# B&R Automation Studio project CombinedLinenSoiledA9KAN (part 8)

#### mnEthInit.st - Initialization code
```iecst
(********************************************************************
 * COPYRIGHT --
 ********************************************************************
 * Program: mnEth
 * File: mnEthInit.st
 * Author: hunholz
 * Created: August 9, 2011
 * Changed: February 3, 2012 2.07.0
 ********************************************************************
 * Implementation of program mnEth
 ********************************************************************)

PROGRAM _INIT

	_xmnEthOk := TRUE;

	_xDHCPstarted := FALSE;
	_xSNTPSrvStarted := FALSE;
	_xSNTPCltStarted := FALSE;

	brsmemset(ADR(kgMsgStatus[MNETH_IDX_KGMSGSTAT]),0,SIZEOF(kgMsgStatus[0]));

	kgMsgStatus[MNETH_IDX_KGMSGSTAT].wFunction_ID := 4;

	// Packet-Version auslesen mit MO_ver aus SYS_lib und für den Additional Status zur Verfügung stellen

	_sPkgName := 'mnEth';

	IF ( MO_ver(ADR(_sPkgName), 0, ADR(_VerStruc)) = 0 ) THEN

		brsmemcpy(ADR(mnEthStatAd.sPkgVersion), ADR(_VerStruc.version), SIZEOF(_VerStruc.version));

	ELSE

		mnEthStatAd.sPkgVersion := '---';

	END_IF

	//***********************************************
	//Lese das Ethernet-Device der CPU aus
	//***********************************************
	REPEAT

		_GetEthPort(enable := TRUE, adrIF := ADR(_sEthDevice));

	UNTIL

		_GetEthPort.status <> ERR_FUB_BUSY

	END_REPEAT

//	brsstrcpy(ADR(_sEthDevice),ADR('IF2'));

		IF brsstrcmp(ADR(_sEthDevice), ADR('ERR')) = 0 THEN

		kgMsgStatus[MNETH_IDX_KGMSGSTAT].wMsgAckLevel := 0;
		kgMsgStatus[MNETH_IDX_KGMSGSTAT].wMsgClass := 10;
		kgMsgStatus[MNETH_IDX_KGMSGSTAT].wMsgNumber := _MENETH_MSG_IFDEVICE;

		_xmnEthOk := FALSE;
		ZANE[1]:= 1;
	END_IF

	//**********************************************************
	//Bestimme den Hostnamen der SPS und setze ihn
	//**********************************************************

	// Adresse von _Info_.InfoGeneral.utfMaschinennummer suchen

//	_xInfoExist := PV_xgetadr(ADR('_Info_.InfoGeneral.utfMaschinennummer'), ADR(_pInfoMaschinennummer), ADR(_lLenInfoMaschinennummer)) = ERR_OK;
//	_xInfoExist := _xInfoExist AND (_lLenInfoMaschinennummer >= 32);

	_xSetDefault := FALSE;

	_CfgGetInaNode(enable := TRUE, pDevice := ADR(_sEthDevice));

	IF _CfgGetInaNode.status = ERR_OK THEN

		IF _CfgGetInaNode.InaNode = 16#FE THEN

			// Setze auf jeden Fall die Default Adresse
			_xSetDefault := TRUE;

		END_IF

	END_IF

	//********************************************************************************************
	//Erzeuge einen Speicherbereich zum parsen oder schreiben von CSV-Dateien
	//********************************************************************************************

	_pParseMem := 0;

	_MemPartCreate(enable := TRUE, len := 512);

	IF _MemPartCreate.status = ERR_OK THEN

		_MemPartAlloc(enable := TRUE, ident := _MemPartCreate.ident, len := 256);

		IF _MemPartAlloc.status = ERR_OK THEN

			_pParseMem := _MemPartAlloc.mem;

		ELSE

			kgMsgStatus[MNETH_IDX_KGMSGSTAT].wMsgAckLevel := 0;
			kgMsgStatus[MNETH_IDX_KGMSGSTAT].wMsgClass := 10;
			kgMsgStatus[MNETH_IDX_KGMSGSTAT].wMsgNumber := _MENETH_MSG_MEM;

			_xmnEthOk := FALSE;
			ZANE[3] := 1;
		END_IF

	ELSE

		kgMsgStatus[MNETH_IDX_KGMSGSTAT].wMsgAckLevel := 0;
		kgMsgStatus[MNETH_IDX_KGMSGSTAT].wMsgClass := 10;
		kgMsgStatus[MNETH_IDX_KGMSGSTAT].wMsgNumber := _MENETH_MSG_MEM;

		_xmnEthOk := FALSE;
	ZANE[2] := 1;

	END_IF

	//**********************************************************
	// Prüfe, ob ein USB-Speicher gesteckt ist
	//**********************************************************

//	_xUSBexist := FALSE;
//
//	IF _xmnEthOk THEN
//
//		_UsbNodeListGet(enable := TRUE, pBuffer := ADR(_NodeIdBuffer), bufferSize := SIZEOF(_NodeIdBuffer), filterInterfaceClass := asusb_CLASS_MASS_STORAGE, filterInterfaceSubClass := 0);
//
//		IF _UsbNodeListGet.status = ERR_OK THEN
//
//			IF _UsbNodeListGet.listNodes > 0 THEN
//
//				_UsbNodeGet(enable := TRUE, nodeId := _NodeIdBuffer[0], pBuffer := ADR(_UsbBufferData), bufferSize := SIZEOF(_UsbBufferData));
//
//				IF _UsbNodeGet.status = ERR_OK THEN
//
//					_sUSBDeviceString := '/DEVICE=';
//					brsstrcpy(ADR(_sUSBDeviceString), ADR(_UsbBufferData.ifName));
//					_xUSBexist := TRUE;
//
//				END_IF
//
//			END_IF
//
//		END_IF
//
//	END_IF

	//******************************************************************************
	// Wenn nicht default gesetzt werden soll, csv-Datei auf USB suchen
	//******************************************************************************

	_xSetIPFromUsb := FALSE;

	IF _xmnEthOk THEN

		IF NOT _xSetDefault THEN

			brsstrcpy(ADR(_sPathCsv), ADR(_sHostname));
			brsstrcat(ADR(_sPathCsv), ADR('\mnEth\mnEth.csv'));

			_FileOpenCsv(enable := TRUE, pDevice := ADR(KG_DEVICE_USBSTICK1), pFile := ADR(_sPathCsv), mode := fiREAD_ONLY);

			IF _FileOpenCsv.status <> ERR_OK THEN

				_FileOpenCsv(enable := TRUE, pDevice := ADR(KG_DEVICE_USBSTICK2), pFile := ADR(_sPathCsv), mode := fiREAD_ONLY);

			END_IF

			IF _FileOpenCsv.status = ERR_OK THEN

				_FileReadCsv(enable := TRUE, ident := _FileOpenCsv.ident, pDest := _pParseMem, len := 256);

				IF _FileReadCsv.status = ERR_OK THEN

					_GetCsvDat.enable := TRUE;
					brwcsncpy( ADR(_GetCsvDat.utfCsvString), _pParseMem+2, 126);
					_GetCsvDat();

					IF _GetCsvDat.RowType = 90 THEN

						brwcsconv(ADR(_ParSetUsb.IP_Adr), ADR(_GetCsvDat.CsvIPRow.utfIP_Adress), 1);
						brwcsconv(ADR(_ParSetUsb.Gateway_Adr), ADR(_GetCsvDat.CsvIPRow.utfGateway), 1);

						IF ethInetAton(pIpStr := ADR(_ParSetUsb.IP_Adr), ADR(_lIPAdr)) = ERR_OK THEN

							IF ethInetAton(pIpStr := ADR(_ParSetUsb.Gateway_Adr), ADR(_lGatewayAdr)) = ERR_OK THEN

								_pOctet ACCESS ADR(_lIPAdr);

								_ParSetUsb.IP_ID1 := _pOctet[0];
								_ParSetUsb.IP_ID2 := _pOctet[1];
								_ParSetUsb.IP_ID3 := (_pOctet[2] / 16) * 16;
								_ParSetUsb.Region := _pOctet[2] MOD 16;
								_ParSetUsb.Station := _pOctet[3];

								IF _ParSetUsb.Region = 3 THEN
									_ParSetUsb.Number := kgGetLineNumberW3(Station := _ParSetUsb.Station, pMachineType := ADR(_kgMachineTypeW3));
								ELSE
									_ParSetUsb.Number := 0;
								END_IF

								// NET-Id bestimmen
								_lNetId := _lIPAdr;
								_pOctet ACCESS ADR(_lNetId);

								_pOctet[2] := _ParSetUsb.IP_ID3;
								_pOctet[3] := 0;

								ethInetNtoa(ipAdr := _lNetId, pIpStr := ADR(_ParSetUsb.NetId_Adr));

								_pOctet ACCESS ADR(_lGatewayAdr);

								_ParSetUsb.GW_ID1 := _pOctet[0];
								_ParSetUsb.GW_ID2 := _pOctet[1];
								_ParSetUsb.GW_ID3 := _pOctet[2];
								_ParSetUsb.GW_ID4 := _pOctet[3];

								_xSetIPFromUsb := TRUE;

							END_IF

						END_IF

					END_IF

				END_IF

				_FileCloseCsv(enable := TRUE, ident := _FileOpenCsv.ident);

			END_IF

//			_sParam := '/DEVICE=';
//			brsstrcat(ADR(_sParam), ADR(_sUSBDeviceString));
//
//			_sUSBDeviceName := 'STICK';
//
//			_DeviceLink(enable := TRUE, pDevice := ADR(_sUSBDeviceName), pParam := ADR(_sParam));
//
//			IF _DeviceLink.status = ERR_OK  AND _pParseMem <> 0 THEN
//
//				_FileOpenCsv(enable := TRUE, pDevice := ADR(_sUSBDeviceName), pFile := ADR(_sPathCsv), mode := fiREAD_ONLY);
//
//				IF _FileOpenCsv.status = ERR_OK THEN
//
//					_FileReadCsv(enable := TRUE, ident := _FileOpenCsv.ident, pDest := _pParseMem, len := 256);
//
//					IF _FileReadCsv.status = ERR_OK THEN
//
//						_GetCsvDat.enable := TRUE;
//						brwcsncpy( ADR(_GetCsvDat.utfCsvString), _pParseMem+2, 126);
//						_GetCsvDat();
//
//						IF _GetCsvDat.RowType = 90 THEN
//
//							brwcsconv(ADR(_ParSetUsb.IP_Adr), ADR(_GetCsvDat.CsvIPRow.utfIP_Adress), 1);
//							brwcsconv(ADR(_ParSetUsb.Gateway_Adr), ADR(_GetCsvDat.CsvIPRow.utfGateway), 1);
//
//							IF ethInetAton(pIpStr := ADR(_ParSetUsb.IP_Adr), ADR(_lIPAdr)) = ERR_OK THEN
//
//								IF ethInetAton(pIpStr := ADR(_ParSetUsb.Gateway_Adr), ADR(_lGatewayAdr)) = ERR_OK THEN
//
//									_pOctet ACCESS ADR(_lIPAdr);
//
//									_ParSetUsb.IP_ID1 := _pOctet[0];
//									_ParSetUsb.IP_ID2 := _pOctet[1];
//									_ParSetUsb.IP_ID3 := (_pOctet[2] / 16) * 16;
//									_ParSetUsb.Region := _pOctet[2] MOD 16;
//									_ParSetUsb.Station := _pOctet[3];
//
//									IF _ParSetUsb.Region = 3 THEN
//										_ParSetUsb.Number := kgGetMachinenumberW3(Station := _ParSetUsb.Station, pMachineType := ADR(_kgMachineTypeW3));
//									ELSE
//										_ParSetUsb.Number := 0;
//									END_IF
//
//									// NET-Id bestimmen
//									_lNetId := _lIPAdr;
//									_pOctet ACCESS ADR(_lNetId);
//
//									_pOctet[2] := _ParSetUsb.IP_ID3;
//									_pOctet[3] := 0;
//
//									ethInetNtoa(ipAdr := _lNetId, pIpStr := ADR(_ParSetUsb.NetId_Adr));
//
//									_pOctet ACCESS ADR(_lGatewayAdr);
//
//									_ParSetUsb.GW_ID1 := _pOctet[0];
//									_ParSetUsb.GW_ID2 := _pOctet[1];
//									_ParSetUsb.GW_ID3 := _pOctet[2];
//									_ParSetUsb.GW_ID4 := _pOctet[3];
//
//									_xSetIPFromUsb := TRUE;
//
//								END_IF
//
//							END_IF
//
//						END_IF
//
//					END_IF
//
//					_FileCloseCsv(enable := TRUE, ident := _FileOpenCsv.ident);
//
//				END_IF
//
//				_DeviceUnlink(enable := TRUE, handle := _DeviceLink.handle);
//
//			END_IF

		END_IF

	END_IF

	//********************************************************************************
	// Sicherstellen, dass das Verzeichnis mnEth auf der CF-Card existiert
	//********************************************************************************

	_DirInfo(enable := TRUE, pDevice := ADR(KG_DEVICE_COMPACTFLASH), pPath := ADR('mnEth'));

	IF _DirInfo.status <> ERR_OK THEN

		_DirCreate(enable := TRUE, pDevice := ADR(KG_DEVICE_COMPACTFLASH), pName := ADR('mnEth'));

	END_IF

	//*****************************************************************************************************
	// Wenn nicht default und nicht von USB gesetzt werden soll, csv-Datei auf CF suchen
	//*****************************************************************************************************

	_xSetIPFromCF := FALSE;

	_sPathCsv := 'mnEth\mnEth.csv';

	IF _xmnEthOk THEN

		IF NOT _xSetDefault  AND NOT _xSetIPFromUsb THEN

			_sPathCsv := 'mnEth\mnEth.csv';

			_FileOpenCsv(enable := TRUE, pDevice := ADR(KG_DEVICE_COMPACTFLASH), pFile := ADR(_sPathCsv), mode := fiREAD_ONLY);

			IF _FileOpenCsv.status = ERR_OK THEN

				_FileReadCsv(enable := TRUE, ident := _FileOpenCsv.ident, pDest := _pParseMem, len := 256);

				IF _FileReadCsv.status = ERR_OK THEN

					_GetCsvDat.enable := TRUE;
					brwcsncpy( ADR(_GetCsvDat.utfCsvString), _pParseMem+2, 126);
					// Nur erste Zeile
					_lPosLF := brwcschr(ADR(_GetCsvDat.utfCsvString),16#0A);
					_lPosCR := brwcschr(ADR(_GetCsvDat.utfCsvString),16#0D);
					IF (_lPosCR <> 0) THEN
						brsmemset(_lPosCR , 0, 2);
					END_IF
					IF (_lPosLF <> 0) THEN
						brsmemset(_lPosLF , 0, 2);
					END_IF

					_GetCsvDat();

					IF _GetCsvDat.RowType = 90 THEN

						brwcsconv(ADR(_ParSetCF.IP_Adr), ADR(_GetCsvDat.CsvIPRow.utfIP_Adress), 1);
						brwcsconv(ADR(_ParSetCF.Gateway_Adr), ADR( _GetCsvDat.CsvIPRow.utfGateway), 1);

						IF ethInetAton(pIpStr := ADR(_ParSetCF.IP_Adr), ADR(_lIPAdr)) = ERR_OK THEN

							IF ethInetAton(pIpStr := ADR(_ParSetCF.Gateway_Adr), ADR(_lGatewayAdr)) = ERR_OK THEN

								_pOctet ACCESS ADR(_lIPAdr);

								_ParSetCF.IP_ID1 := _pOctet[0];
								_ParSetCF.IP_ID2 := _pOctet[1];
								_ParSetCF.IP_ID3 := (_pOctet[2] / 16) * 16;
								_ParSetCF.Region := _pOctet[2] MOD 16;
								_ParSetCF.Station := _pOctet[3];

								IF _ParSetCF.Region = 3 THEN
									_ParSetCF.Number := kgGetLineNumberW3(Station := _ParSetCF.Station, pMachineType := ADR(_kgMachineTypeW3));
								ELSE
									_ParSetCF.Number := 0;
								END_IF

								// NET-Id bestimmen
								_lNetId := _lIPAdr;
								_pOctet ACCESS ADR(_lNetId);

								_pOctet[2] := _ParSetCF.IP_ID3;
								_pOctet[3] := 0;

								ethInetNtoa(ipAdr := _lNetId, pIpStr := ADR(_ParSetCF.NetId_Adr));

								_pOctet ACCESS ADR(_lGatewayAdr);

								_ParSetCF.GW_ID1 := _pOctet[0];
								_ParSetCF.GW_ID2 := _pOctet[1];
								_ParSetCF.GW_ID3 := _pOctet[2];
								_ParSetCF.GW_ID4 := _pOctet[3];

								_xSetIPFromCF := TRUE;

							END_IF

						END_IF

					END_IF

				END_IF

				_FileCloseCsv(enable := TRUE, ident := _FileOpenCsv.ident);

			END_IF

		END_IF

	END_IF

	//*****************************************************************************************************
	// Adressen von CF oder USB setzen
	//*****************************************************************************************************

	IF _xmnEthOk THEN

		IF _xSetIPFromCF OR _xSetIPFromUsb THEN

			IF _xSetIPFromCF THEN
				_ParSet := _ParSetCF;
			ELSE
				_ParSet := _ParSetUsb;
			END_IF

// Für Testzwecke in Hausnetzen mit anderer Netzwerkmaske

#ifndef NoSubnetMask

			_CfgGetSubnetMask(enable := TRUE, pDevice := ADR(_sEthDevice), pSubnetMask := ADR(_sActSubnetMask), Len := SIZEOF(_sActSubnetMask));

			IF (brsstrcmp(ADR(_sActSubnetMask), ADR(_sSubnetMask)) <> 0) THEN

				_CfgSetSubnetMask(enable := TRUE, pDevice := ADR(_sEthDevice), pSubnetMask := ADR(_sSubnetMask), Option := cfgOPTION_NON_VOLATILE);

			END_IF
#endif
			_pOctet ACCESS ADR(_lBroadcastAdr);

			_pOctet[0] := _ParSet.IP_ID1;
			_pOctet[1] := _ParSet.IP_ID2;
			_pOctet[2] := _ParSet.IP_ID3 + 15;
			_pOctet[3] := 255;

			ethInetNtoa(ADR(_lBroadcastAdr), ADR(_sBroadcastAdr));

			_CfgGetBroadcastAdr(enable := TRUE, pDevice := ADR(_sEthDevice), pBroadcastAddr := ADR(_sActBroadcastAdr), Len := SIZEOF(_sActBroadcastAdr));

			IF (brsstrcmp(ADR(_sActBroadcastAdr), ADR(_sBroadcastAdr)) <> 0) THEN

				_CfgSetBroadcastAdr(enable := TRUE, pDevice := ADR(_sEthDevice), pBroadcastAddr := ADR(_sBroadcastAdr), Option := cfgOPTION_NON_VOLATILE);

			END_IF

			_CfgGetIPAddress(enable := TRUE, pDevice := ADR(_sEthDevice), pIPAddr := ADR(_sActIPAdr), Len := SIZEOF(_sActIPAdr));

			IF (brsstrcmp(ADR(_sActIPAdr), ADR(_ParSet.IP_Adr)) <> 0) THEN

				_CfgSetIPAddr(enable := TRUE, pDevice := ADR(_sEthDevice), pIPAddr := ADR(_ParSet.IP_Adr), Option := cfgOPTION_NON_VOLATILE);

			END_IF

			_CfgGetGateway(enable := TRUE, pDevice := ADR(_sEthDevice), pGateway := ADR(_sActGateway), Len := SIZEOF(_sActGateway));

			IF (brsstrcmp(ADR(_sActGateway), ADR(_ParSet.Gateway_Adr)) <> 0) THEN

				_CfgSetDefaultGateway(enable := TRUE, pDevice := ADR(_sEthDevice), pGateway := ADR(_ParSet.Gateway_Adr), Option := cfgOPTION_NON_VOLATILE);

			END_IF

			_ParAktuell := _ParSet;

		ELSE

			_CfgGetGateway(enable := TRUE, pDevice := ADR(_sEthDevice), pGateway := ADR(_ParAktuell.Gateway_Adr), Len := SIZEOF(_ParAktuell.Gateway_Adr));

			_CfgGetIPAddress(enable := TRUE, pDevice := ADR(_sEthDevice), pIPAddr := ADR(_ParAktuell.IP_Adr), Len := SIZEOF(_ParAktuell.IP_Adr));

			IF ethInetAton(pIpStr := ADR(_ParAktuell.IP_Adr), ADR(_lIPAdr)) = ERR_OK THEN

				IF ethInetAton(pIpStr := ADR(_ParAktuell.Gateway_Adr), ADR(_lGatewayAdr)) = ERR_OK THEN

					_pOctet ACCESS ADR(_lIPAdr);

					_ParAktuell.IP_ID1 := _pOctet[0];
					_ParAktuell.IP_ID2 := _pOctet[1];
					_ParAktuell.IP_ID3 := (_pOctet[2] / 16) * 16;
					_ParAktuell.Region := _pOctet[2] MOD 16;
					_ParAktuell.Station := _pOctet[3];

					IF _ParAktuell.Region = 3 THEN
						_ParAktuell.Number := kgGetLineNumberW3(Station := _ParAktuell.Station, pMachineType := ADR(_kgMachineTypeW3));
					ELSE
						_ParAktuell.Number := 0;
					END_IF

					// NET-Id bestimmen
					_lNetId := _lIPAdr;
					_pOctet ACCESS ADR(_lNetId);

					_pOctet[2] := _ParAktuell.IP_ID3;
					_pOctet[3] := 0;

					ethInetNtoa(ipAdr := _lNetId, pIpStr := ADR(_ParAktuell.NetId_Adr));

					_pOctet ACCESS ADR(_lGatewayAdr);

					_ParAktuell.GW_ID1 := _pOctet[0];
					_ParAktuell.GW_ID2 := _pOctet[1];
					_ParAktuell.GW_ID3 := _pOctet[2];
					_ParAktuell.GW_ID4 := _pOctet[3];

				END_IF

			END_IF

		END_IF

		IF NOT _xSetIPFromCF AND NOT _xSetIPFromUsb THEN

			_xSetDefault := TRUE;

		END_IF

		_xChanged := FALSE;

	END_IF

	//*****************************************************************************************************
	// CSV-Datei schreiben, wenn Daten vom USB gekommen sind
	//*****************************************************************************************************

	IF _xmnEthOk THEN

		IF _xSetIPFromUsb OR NOT _xSetIPFromCF THEN

			brsmemset(_pParseMem, 0, 256);

			_lFileSize := 0;

			brwcsconv(ADR( _IPRow.utfIP_Adress), ADR(_ParAktuell.IP_Adr), 0);
			brwcsconv(ADR(_IPRow.utfGateway), ADR(_ParAktuell.Gateway_Adr), 0);

			_WriteBOM(enable := TRUE, pMem := _pParseMem, lMaxSize := 256, lSize := _lFileSize);
			_WriteCsv90(enable := TRUE, pMem := _pParseMem, lMaxSize := 256, IPRow := _IPRow, lSize := _lFileSize);

			_FileDeleteCsv(enable := TRUE, pDevice := ADR(KG_DEVICE_COMPACTFLASH), pName := ADR(_sPathCsv));

			_FileCreateCsv(enable := TRUE, pDevice := ADR(KG_DEVICE_COMPACTFLASH), pFile := ADR(_sPathCsv));

			_FileOpenCsv(enable := TRUE, pDevice := ADR(KG_DEVICE_COMPACTFLASH), pFile := ADR(_sPathCsv), mode := fiWRITE_ONLY);

			IF _FileOpenCsv.status = ERR_OK THEN

				_FileWriteCsv(enable := TRUE, ident := _FileOpenCsv.ident, offset := 0, pSrc := _pParseMem, len := _lFileSize);

				_FileCloseCsv(enable := TRUE, ident := _FileOpenCsv.ident);

			END_IF

		END_IF

	END_IF

END_PROGRAM
```

#### mnEth.typ - Local data types
```iecst
(********************************************************************
 * COPYRIGHT --
 ********************************************************************
 * Program: mnEth
 * File: mnEth.typ
 * Author: tamme
 * Created: March 17, 2011
 ********************************************************************
 * Local data types of program mnEth
 ********************************************************************)

TYPE
	enumEthernetState :
		(
		es_idle := 0,
		es_SetDef1 := 100,
		es_SetDef2,
		es_SetDef3,
		es_SetDef4,
		es_SetDef5,
		es_WriteCSV1 := 200,
		es_WriteCSV2,
		es_WriteCSV3,
		es_WriteCSV4,
		es_WriteCSV5,
		es_WriteCSV6,
		es_Change1 := 300,
		es_Change2,
		es_Change3,
		es_Change4,
		es_Change5,
		es_Change6,
		es_Change7,
		es_DHCP1 := 400,
		es_DHCP2,
		es_DHCP3,
		es_SNTPcltStart1 := 500,
		es_SNTPcltStop1 := 510,
		es_SNTPsrvStart1 := 520,
		es_SNTPsrvStop1 := 530,
		es_SetHostname1 := 600,
		es_SetHostname2,
		es_SetHostname3,
		es_Warning := 900
		);
	_EthPar_typ : 	STRUCT
		IP_ID1 : USINT;
		IP_ID2 : USINT;
		IP_ID3 : USINT;
		Region : USINT;
		Station : USINT;
		Number : USINT;
		GW_ID1 : USINT;
		GW_ID2 : USINT;
		GW_ID3 : USINT;
		GW_ID4 : USINT;
		IP_Adr : STRING[15];
		Gateway_Adr : STRING[15];
		NetId_Adr : STRING[15];
	END_STRUCT;
END_TYPE
```

#### mnEth.var - Local variables
```iecst
(********************************************************************
 * COPYRIGHT --
 ********************************************************************
 * Program: mnEth
 * File: mnEth.var
 * Author: tamme
 * Created: March 17, 2011
 * Changed: September 20, 2011
 ********************************************************************
 * Local variables of program mnEth
 ********************************************************************)
VAR
	_xmnEthOk : BOOL;
END_VAR
(*Ermittlung des Ethernetinterface*)
VAR
	_GetEthPort : kgGetEthPort;
	_sEthDevice : STRING[15];
END_VAR
(*Maschinennummer*)
VAR
	_sMnr : STRING[15];
END_VAR
(*Hostname*)
VAR
	_CfgSetHostName : CfgSetHostName;
	_sHostname : STRING[15];
END_VAR
(*Defaultwerte setzen*)
VAR
	_xSetDefault : BOOL;
END_VAR
(*Werte vom USB*)
VAR
	_ParSetUsb : _EthPar_typ;
	_FileOpenCsv : FileOpen;
	_xSetIPFromUsb : BOOL;
END_VAR
(*Parsen allgemein*)
VAR
	_sPathCsv : STRING[127];
	_MemPartCreate : AsMemPartCreate;
	_MemPartAlloc : AsMemPartAlloc;
	_pParseMem : UDINT;
	_FileReadCsv : FileRead;
	_FileCloseCsv : FileClose;
	_GetCsvDat : mnParam_GetCsvDat;
	_lFileSize : UDINT;
END_VAR
(*Hilfsvariablen*)
VAR
	_ParSet : _EthPar_typ;
	_lIPAdr : UDINT;
	_pOctet : REFERENCE TO ARRAY[0..3] OF USINT;
	_lGatewayAdr : UDINT;
	_DirInfo : DirInfo;
	_DirCreate : DirCreate;
	_lBroadcastAdr : UDINT;
	_sBroadcastAdr : STRING[15];
	_xChanged : BOOL;
END_VAR
(*Werte von CF*)
VAR
	_ParSetCF : _EthPar_typ;
	_xSetIPFromCF : BOOL;
END_VAR
(*Funktionen*)
VAR
	_CfgSetSubnetMask : CfgSetSubnetMask;
	_CfgSetIPAddr : CfgSetIPAddr;
	_CfgSetDefaultGateway : CfgSetDefaultGateway;
	_CfgSetBroadcastAdr : CfgSetBroadcastAddr;
	_CfgGetGateway : CfgGetDefaultGateway;
	_CfgGetIPAddress : CfgGetIPAddr;
END_VAR
(*Werte schreiben*)
VAR
	_WriteBOM : mnParam_WriteBOM_Mem;
	_WriteCsv90 : mnParam_WriteCSV90_Mem;
	_IPRow : mnParam_CsvIPRow_typ;
	_FileDeleteCsv : FileDelete;
	_FileCreateCsv : FileCreate;
	_FileWriteCsv : FileWrite;
END_VAR
(*Zyklisch*)
VAR
	_ParGet : _EthPar_typ;
	_ParAktuell : _EthPar_typ;
	enEState : enumEthernetState;
	_TONidle : TON;
	_TONwarning : TON;
	_bWaitCounter : USINT;
END_VAR
(*Konstanten*)
VAR CONSTANT
	_MENETH_MSG_IFDEVICE : UINT := 20000;
	_MENETH_MSG_MEM : UINT := 20001;
	_MENETH_MSG_SETDEF : UINT := 20100;
	_MENETH_MSG_WRITECSV : UINT := 20101;
	_MENETH_MSG_CHANGE : UINT := 20102;
END_VAR
VAR
	_CfgGetInaNode : CfgGetInaNode;
	_lPosLF : UDINT;
	_lPosCR : UDINT;
	_kgMachineTypeW3 : kgMachinetypeW3_typ;
	_lNetId : UDINT;
	_cfgLease : cfgLease_typ;
	_CfgSetDhcpsData : CfgSetDhcpsData;
	_xDHCPstarted : BOOL;
	_CfgSetDhcpServer : CfgSetDhcpServer;
	_xSNTPSrvStarted : BOOL;
	_xSNTPCltStarted : BOOL;
	_CfgSetSntpClient : CfgSetSntpClient;
	_CfgSetSntpServer : CfgSetSntpServer;
	_sSubnetMask : STRING[15] := '255.255.240.000';
	_xSetHostname : BOOL := TRUE;
	_CfgGetHostName : CfgGetHostName;
	_sActHostname : STRING[15];
	_CfgGetSubnetMask : CfgGetSubnetMask;
	_sActSubnetMask : STRING[15];
	_CfgGetBroadcastAdr : CfgGetBroadcastAddr;
	_sActBroadcastAdr : STRING[15];
	_sActIPAdr : STRING[15];
	_sActGateway : STRING[15];
	_sPkgName : STRING[11];
	_VerStruc : MoVerStruc_typ;
	_kgMsgStatus : kgMsg_Status_Typ;
	ZANE : ARRAY[0..5] OF BOOL;
END_VAR
```

### Pkg_mnEth_History.txt
```
2.01.0	2011-09-07	AH Änderung der Standardnetzwerkmaske auf 20 bit
2.02.0	2011-09-20	AH Schaut jetzt auf mnParamStatAd.xParamOK, setzt Version 0.5 von mnParam voraus
2.02.1	2011-09-28	AH Interface für PCTs korregiert
2.03.0	2011-10-06	AH Maschinennummer aus _Info_, IP-Adresse usw. NONVOLATILE
2.04.0	2011-10-20	AH Umstellung auf AS 3.0.90
2.05.0	2012-01-10	AH PackageVersion wird nun in mnEthStatAd angezeigt
2.06.0	2012-01-27	AH Unabhängig von NetLink
2.07.0	2012-02-03	AH Es wird kein USB-Stick mehr als Device gelinkt. Es wird vorausgesetzt, dass die
					   Devices (Siehe Konstanten KG_DEVICE_USBSTICK1 und KG_DEVICE_USBSTICK2 bereits
					   in der sysconf festgelegt sind) Setzt KGStandard 1.14.0 voraus.
2.08.0	2012-02-08	AH Kompatibel zu KGStandard 1.15.0 (KGstdLib 1.03.0)
2.09.0	2012-02-23	AH Kompatibel zu hlKanLink 0.94.0
					   - Hostname auf 15 Zeichen gekürzt
					   Kompatibel mit mnTest
2.09.1	2012-03-20	AH Abhängigkeiten ergänzt
```

### Package Logical/Mewa/KGFramework/Pkg_mnCnt - Management-Ebene für Zähler

### Pkg_mnCnt.typ - Global data types
```iecst
(********************************************************************
 * COPYRIGHT -- Microsoft
 ********************************************************************
 * Package: Pkg_mnCnt
 * File: Pkg_mnCnt.typ
 * Author: hunholz
 * Created: July 02, 2011
 ********************************************************************
 * Data types of package Pkg_mnCnt
 ********************************************************************)

TYPE
	mnCntLocation_Typ : 	STRUCT
		sNameId : STRING[10]; (*Text-ID des Ortes*)
		bLocationExt : USINT; (*0 - Interner Ort, 1 - Externer Ort*)
	END_STRUCT;
	mnCntStatAd_Typ : 	STRUCT
		sPkgVersion : STRING[10];
	END_STRUCT;
	mnCntEventBatch_Typ : 	STRUCT
		Batch : BatchData_typ;
		FromLocation : mnCntLocation_Typ;
		ToLocation : mnCntLocation_Typ;
		bProgram : USINT;
		bEvent : USINT; (*0 - Beladung, 1 - Entladung, 2 - Geändert, 3 - Gelöscht*)
	END_STRUCT;
	mnCntEventCounter_Typ : 	STRUCT
		Source : mnCntLocation_Typ; (*Quell Ort für Medien*)
		Destination : mnCntLocation_Typ; (*Ziel Ort für Medien, Ort der Messung*)
		BatchNo : GUID_type; (*Postennummer (long oder GUID)*)
		dtTimeStamp : DATE_AND_TIME; (*Zeitstempel des Zählwerts*)
		lAmount : UDINT; (*Menge bzw. Wert*)
		lNomAmount : UDINT; (*Sollmenge*)
		bTypeBatchNo : USINT; (*0 - Postennummer ist long, 1 - Postennummer ist GUID*)
		bType : USINT; (*1 - Wasser, 2 - Dampf, 3 - Gas, 4 - Elektrische Energie, 11 - Temperatur, 12 - Druck, 13 - Drehzahl*)
	END_STRUCT;
	mnCntEventDosing_Typ : 	STRUCT
		BatchNo : GUID_type; (*Postennummer (long oder GUID)*)
		dtTimeStamp : DATE_AND_TIME; (*Zeitstempel der Dosierung*)
		rNomAmount : REAL; (*Solldosiermenge*)
		rAmount : REAL; (*Istdosiermenge*)
		rPumpConst : REAL; (*Pumpenkonstante*)
		sUnit : STRING[11]; (*Einheit der Dosierung*)
		utfName : WSTRING[23]; (*Name der Dosierung*)
		Source : mnCntLocation_Typ; (*Quelle*)
		Destination : mnCntLocation_Typ; (*Zielort*)
		bTypeBatchNo : USINT; (*0 - Postennummer ist long, 1 - Postennummer ist GUID*)
	END_STRUCT;
	mnCntEventDosingId_Typ : 	STRUCT
		bId : USINT;
		DosingEvent : mnCntEventDosing_Typ;
	END_STRUCT;
	mnCntEventTime_Typ : 	STRUCT
		dtTimeStamp : DATE_AND_TIME;
		lAmount : UDINT; (*Zeitintervall*)
		bState : USINT; (*0 - Inaktiv, 1 - Warten, 2 - Aktiv*)
		bSubState : USINT; (*0.0 - AUS/Taktende, 0.1 - Stop, 0.2 - int. Störung, 0.3 - ext. Störung, 0.4 - Sicherer Halt, 0.5 - NOT-HALT, 1.0 - Beladung, 1.1 - Entladung, 1.2 - Dosierung, 2.0 - Prozess, 2.1 - Vorbereitung*)
	END_STRUCT;
	IFmnCntOut_Typ : 	STRUCT
		wStatus : UINT;
		xBatchEventReadOK : BOOL;
		xCounterEventReadOK : ARRAY[0..MNCNT_IDX_COUNTER_MAX]OF BOOL;
		xDosingEventReadOK : ARRAY[1..48]OF BOOL;
		xTimeEventReadOK : BOOL;
	END_STRUCT;
	IFmnCntIn_Typ : 	STRUCT
		wCmd : UINT;
		bBatchEventValid : USINT; (*0->1: Batchevent übernehmen*)
		bCntEventValid : ARRAY[0..MNCNT_IDX_COUNTER_MAX]OF USINT; (*0->1 : Zählerwert übernehmen*)
		bDosingEventValid : ARRAY[1..48]OF USINT; (*0->1 : Zählerwert übernehmen*)
		bTimeEventValid : USINT; (*0->1 : Zeitwert übernehmen*)
		BatchEvent : mnCntEventBatch_Typ; (*Postenevent*)
		CounterEvent : ARRAY[0..MNCNT_IDX_COUNTER_MAX]OF mnCntEventCounter_Typ; (*Zählerevents*)
		DosingEvent : ARRAY[1..48]OF mnCntEventDosing_Typ; (*max. 48 Dosierevents*)
		TimeEvent : mnCntEventTime_Typ; (*Zeitwerte*)
	END_STRUCT;
	IFmnCnt_Typ : 	STRUCT
		In : IFmnCntIn_Typ;
		Out : IFmnCntOut_Typ;
	END_STRUCT;
	mnCntParMacDosingDef_Typ : 	STRUCT
		utfName : WSTRING[23];
		xUseConversion : BOOL;
		bCompartment : USINT;
		bIdx : USINT;
		bReserve : USINT;
		rConversionMultiplier : REAL;
		sUnit : STRING[11];
	END_STRUCT;
	mnCntParMac_Typ : 	STRUCT
		DosingDefines : ARRAY[1..48]OF mnCntParMacDosingDef_Typ;
	END_STRUCT;
	mnCntPar_Typ : 	STRUCT
		Mac : mnCntParMac_Typ;
	END_STRUCT;
END_TYPE
```

### Pkg_mnCnt.var - Global variables
```iecst
(********************************************************************
 * COPYRIGHT -- Microsoft
 ********************************************************************
 * Package: Pkg_mnCnt
 * File: Pkg_mnCnt.var
 * Author: hunholz
 * Created: July 02, 2011
 ********************************************************************
 * Variables of package Pkg_mnCnt
 ********************************************************************)
VAR
	IFmnCnt : IFmnCnt_Typ := (0);
	mnCntCmd : KG_Cmd_typ := (0);
	mnCntPar : mnCntPar_Typ := (0);
	mnCntStatAd : mnCntStatAd_Typ;
END_VAR
(*Konstanten*)
VAR CONSTANT
	MNCNT_MSG_READ_SUM : UINT := 1000;
	MNCNT_MSG_DELETE_SUM : UINT := 1001;
	MNCNT_MSG_CREATE_SUM : UINT := 1002;
	MNCNT_MSG_INFO_SUM : UINT := 1003;
	MNCNT_MSG_CREATE_RB : UINT := 1004;
	MNCNT_MSG_INFO_RB : UINT := 1005;
	MNCNT_MSG_CFG : UINT := 1006;
	MNCNT_MSG_CNT_CFG : UINT := 1007;
	MNCNT_MSG_RB_NEW : UINT := 1009;
	MNCNT_BATCHEVENT_LOAD : USINT := 0; (*Postenevent bei Beladung*)
	MNCNT_BATCHEVENT_UNLOAD : USINT := 1; (*Postenevent bei Entladung*)
	MNCNT_BATCHEVENT_CHANGEDATA : USINT := 2; (*Postenevent bei Datenänderung*)
	MNCNT_BATCHEVENT_DELETE : USINT := 3; (*Postenevent zum Löschen eines Postens*)
	MNCNT_COUNTERTYPE_WATER : USINT := 1; (*Wasserzähler*)
	MNCNT_COUNTERTYPE_STEAM : USINT := 2; (*Dampf*)
	MNCNT_COUNTERTYPE_GAS : USINT := 3; (*Gas*)
	MNCNT_COUNTERTYPE_ELECTRICENERGY : USINT := 4; (*Elektrische Energie*)
	MNCNT_COUNTERTYPE_NOTCOUNTABLE : USINT := 11; (*Nicht zählbare Werte*)
	MNCNT_COUNTERTYPE_TEMPERATURE : USINT := 11; (*Temperatur*)
	MNCNT_COUNTERTYPE_PRESSURE : USINT := 12; (*Druck*)
	MNCNT_COUNTERTYPE_RPM : USINT := 13; (*Drehzahl*)
	MNCNT_IDX_TIMESTATE_MAX : UINT := 2; (*0 - PAUSED, 1 - WAIT, 2 - ACTIVE*)
	MNCNT_TIMERSTATE_PAUSED : USINT := 0;
	MNCNT_TIMERSTATE_WAIT : USINT := 1;
	MNCNT_TIMERSTATE_ACTIVE : USINT := 2;
	MNCNT_IDX_TIMESUBSTATE_MAX : UINT := 6;
	MNCNT_TIMERSUBSTATE_WASHING : USINT := 0;
	MNCNT_TIMERSUBSTATE_PREPERATION : USINT := 1;
	MNCNT_TIMERSUBSTATE_TRANSFER : USINT := 2;
	MNCNT_TIMERSUBSTATE_PREPFORSTOP : USINT := 3;
	MNCNT_TIMERSUBSTATE_LOADING : USINT := 0;
	MNCNT_TIMERSUBSTATE_UNLOADING : USINT := 1;
	MNCNT_TIMERSUBSTATE_DOSING : USINT := 2;
	MNCNT_TIMERSUBSTATE_WATERLEVEL : USINT := 3;
	MNCNT_TIMERSUBSTATE_TEMPERATURE : USINT := 4;
	MNCNT_TIMERSUBSTATE_DISINFECTION : USINT := 5;
	MNCNT_TIMERSUBSTATE_AIRPRESSURE : USINT := 6;
	MNCNT_TIMERSUBSTATE_OFF : USINT := 0;
	MNCNT_TIMERSUBSTATE_STOP : USINT := 1;
	MNCNT_TIMERSUBSTATE_INTFAULT : USINT := 2;
	MNCNT_TIMERSUBSTATE_EXTFAULT : USINT := 3;
	MNCNT_TIMERSUBSTATE_SAFESTOP : USINT := 4;
	MNCNT_TIMERSUBSTATE_EMERGENCYSTP : USINT := 5;
END_VAR
```

- Program Logical/Mewa/KGFramework/Pkg_mnCnt/mnCnt (IEC) - Counter Manager (no source held here)

### Package Logical/Mewa/KGFramework/Pkg_mnMsg - Meldungs-Manager

### Program Logical/Mewa/KGFramework/Pkg_mnMsg/mnMsg (IEC) - Meldungsmanager
